FUNCTION_BLOCK VALUES_TO_JSON
  {SET_ATTRIBUTE(OpcUa, SERVICE)}
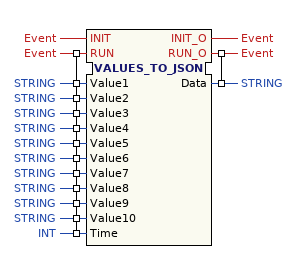
  EVENT_INPUT
    INIT;
    RUN WITH Value1, Value2, Value3, Value4, Value5, Value6, Value7, Value8, Value9, Value10, Time; {SET_ATTRIBUTE(OpcUa, Method)}
  END_EVENT
  EVENT_OUTPUT
    INIT_O;
    RUN_O WITH Data;
  END_EVENT
  VAR_INPUT
    Value1 : STRING; {SET_ATTRIBUTE(OpcUa, Variable.RUN)}
    Value2 : STRING; {SET_ATTRIBUTE(OpcUa, Variable.RUN)}
    Value3 : STRING; {SET_ATTRIBUTE(OpcUa, Variable.RUN)}
    Value4 : STRING; {SET_ATTRIBUTE(OpcUa, Variable.RUN)}
    Value5 : STRING; {SET_ATTRIBUTE(OpcUa, Variable.RUN)}
    Value6 : STRING; {SET_ATTRIBUTE(OpcUa, Variable.RUN)}
    Value7 : STRING; {SET_ATTRIBUTE(OpcUa, Variable.RUN)}
    Value8 : STRING; {SET_ATTRIBUTE(OpcUa, Variable.RUN)}
    Value9 : STRING; {SET_ATTRIBUTE(OpcUa, Variable.RUN)}
    Value10 : STRING; {SET_ATTRIBUTE(OpcUa, Variable.RUN)}
    Time : INT; {SET_ATTRIBUTE(OpcUa, Variable.RUN)}
  END_VAR
  VAR_OUTPUT
    Data : STRING; {SET_ATTRIBUTE(OpcUa, Variable.RUN)}
  END_VAR
END_FUNCTION_BLOCK
